# EPICS autosave request: urRobotApp/Db/waypoint_action_settings.req
file calcout_settings.req P=$(P)ActionDoneCalc$(N)
file yySseq_settings.req P=$(P),S=ActionSseq$(N)
